INTERFACE I_DriveBase

METHOD Disable : BOOL
VAR_INPUT
END_VAR
END_METHOD

METHOD Enable : BOOL
VAR_INPUT
END_VAR
END_METHOD

END_INTERFACE

(* stored: Version 1.1.0.1
   Itf I_DriveBase: Id {5128345e-1585-4387-9646-8862db27e221}
   Method Disable: Id {fc485f0e-5ed1-49ff-a430-f767fedfa7cf}
   Method Enable: Id {b4d05e17-2285-4c6e-a1de-f86c09305f4b} *)
